// TIA Portal V19 export
FUNCTION "NEW_FUNCTION" : Void   // FC2, LAD
TITLE = New Function Added
{ S7_Optimized_Access := 'TRUE' }
// stored: SetENOAutomatically false
BEGIN

REGION Network 1: New Function 1
   // Testing adding a new function.
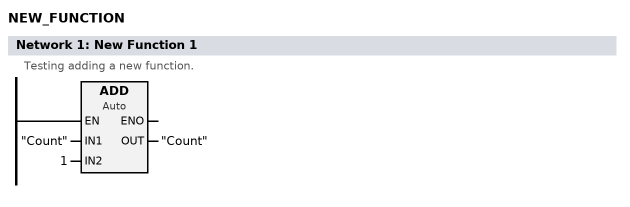
   RUNG wire#powerrail
      Add(in1 := "Count", in2 := 1, out => "Count")
   END_RUNG
   // the same network as SCL:
   "Count" := "Count" + 1;
END_REGION
END_FUNCTION
